ABB RobotStudio station: Box Sorting by Size v1.rspag

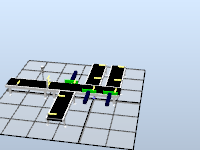
Station Box Sorting by Size v1 (saved by RobotStudio 21.4.9700.0)
Layout (positions relative to the parent item):
  - SUB010 [protected smart component, left out]
  - SUB020 [protected smart component, left out]
  - SUB050 [protected smart component, left out]
  - SUB040 [protected smart component, left out]
  - SUB030 [protected smart component, left out]
  - ProductInput [protected smart component, left out]
  - SUB600LightBeacon [protected smart component, left out]
  - OpcUaClient [smart component, from Components\OpcUaClient.rslib]
      properties: Status=Disconnected; ServerAddress=opc.tcp://localhost:4840; UseSecurity=false; AutoConnect=false; SignalConfiguration=NamespaceUri;IdentifierType;Identifier;ReadWrite;Signal;SignalType;Controller;Device
CODESYSSPV3/3S/IecVarAccess;String;|var|CODESYS Control Win V3 x64.Application.IOs.iSUB010_B1;Write;iSUB010_B1;Digital;;
CODESYSSPV3/3S/IecVarAccess;String;|var|CODESYS Control Win V3 x64.Application.IOs.iSUB010_B2;Write;iSUB010_B2;Digital;;
CODESYSSPV3/3S/IecVarAccess;String;|var|CODESYS Control Win V3 x64.Application.IOs.iSUB010_B3;Write;iSUB010_B3;Digital;;
CODESYSSPV3/3S/IecVarAccess;String;|var|CODESYS Control Win V3 x64.Application.IOs.iSUB010_B4;Write;iSUB010_B4;Digital;;
CODESYSSPV3/3S/IecVarAccess;String;|var|CODESYS Control Win V3 x64.Application.IOs.iSUB020_B1;Write;iSUB020_B1;Digital;;
CODESYSSPV3/3S/IecVarAccess;String;|var|CODESYS Control Win V3 x64.Application.IOs.iSUB020_B2;Write;iSUB020_B2;Digital;;
CODESYSSPV3/3S/IecVarAccess;String;|var|CODESYS Control Win V3 x64.Application.IOs.iSUB020_B3;Write;iSUB020_B3;Digital;;
CODESYSSPV3/3S/IecVarAccess;String;|var|CODESYS Control Win V3 x64.Application.IOs.iSUB030_B1;Write;iSUB030_B1;Digital;;
CODESYSSPV3/3S/IecVarAccess;String;|var|CODESYS Control Win V3 x64.Application.IOs.iSUB030_B2;Write;iSUB030_B2;Digital;;
CODESYSSPV3/3S/IecVarAccess;String;|var|CODESYS Control Win V3 x64.Application.IOs.iSUB030_C1_B1;Write;iSUB030_C1_B1;Digital;;
CODESYSSPV3/3S/IecVarAccess;String;|var|CODESYS Control Win V3 x64.Application.IOs.iSUB040_B1;Write;iSUB040_B1;Digital;;
CODESYSSPV3/3S/IecVarAccess;String;|var|CODESYS Control Win V3 x64.Application.IOs.iSUB040_B2;Write;iSUB040_B2;Digital;;
CODESYSSPV3/3S/IecVarAccess;String;|var|CODESYS Control Win V3 x64.Application.IOs.iSUB040_C1_B1;Write;iSUB040_C1_B1;Digital;;
CODESYSSPV3/3S/IecVarAccess;String;|var|CODESYS Control Win V3 x64.Application.IOs.iSUB050_B1;Write;iSUB050_B1;Digital;;
CODESYSSPV3/3S/IecVarAccess;String;|var|CODESYS Control Win V3 x64.Application.IOs.iSUB050_B2;Write;iSUB050_B2;Digital;;
CODESYSSPV3/3S/IecVarAccess;String;|var|CODESYS Control Win V3 x64.Application.IOs.iSUB050_C1_B1;Write;iSUB050_C1_B1;Digital;;
CODESYSSPV3/3S/IecVarAccess;String;|var|CODESYS Control Win V3 x64.Application.IOs.oSUB000_H4;Read;oSUB000_H4;Digital;;
CODESYSSPV3/3S/IecVarAccess;String;|var|CODESYS Control Win V3 x64.Application.IOs.oSUB000_H5;Read;oSUB000_H5;Digital;;
CODESYSSPV3/3S/IecVarAccess;String;|var|CODESYS Control Win V3 x64.Application.IOs.oSUB000_H6;Read;oSUB000_H6;Digital;;
CODESYSSPV3/3S/IecVarAccess;String;|var|CODESYS Control Win V3 x64.Application.IOs.oSUB010_K1;Read;oSUB010_K1;Digital;;
CODESYSSPV3/3S/IecVarAccess;String;|var|CODESYS Control Win V3 x64.Application.IOs.oSUB020_K1;Read;oSUB020_K1;Digital;;
CODESYSSPV3/3S/IecVarAccess;String;|var|CODESYS Control Win V3 x64.Application.IOs.oSUB030_K1;Read;oSUB030_K1;Digital;;
CODESYSSPV3/3S/IecVarAccess;String;|var|CODESYS Control Win V3 x64.Application.IOs.oSUB030_Y1;Read;oSUB030_Y1;Digital;;
CODESYSSPV3/3S/IecVarAccess;String;|var|CODESYS Control Win V3 x64.Application.IOs.oSUB040_K1;Read;oSUB040_K1;Digital;;
CODESYSSPV3/3S/IecVarAccess;String;|var|CODESYS Control Win V3 x64.Application.IOs.oSUB040_Y1;Read;oSUB040_Y1;Digital;;
CODESYSSPV3/3S/IecVarAccess;String;|var|CODESYS Control Win V3 x64.Application.IOs.oSUB050_K1;Read;oSUB050_K1;Digital;;
CODESYSSPV3/3S/IecVarAccess;String;|var|CODESYS Control Win V3 x64.Application.IOs.oSUB050_Y1;Read;oSUB050_Y1;Digital;;

  - SUB030Cylinder [protected smart component, left out]
  - SUB040Cylinder [protected smart component, left out]
  - SUB050Cylinder [protected smart component, left out]
  - Sensors [graphiccomponentgroup]
    - SUB010_B1 [protected smart component, left out]
    - SUB020_B1 [protected smart component, left out]
    - SUB020_B2 [protected smart component, left out]
    - SUB020_B3 [protected smart component, left out]
    - SUB030_B1 [protected smart component, left out]
    - SUB030_B2 [protected smart component, left out]
    - SUB040_B1 [protected smart component, left out]
    - SUB040_B2 [protected smart component, left out]
    - SUB050_B1 [protected smart component, left out]
    - SUB050_B2 [protected smart component, left out]
    - SUB010_B2 [protected smart component, left out]
    - SUB010_B3 [protected smart component, left out]
    - SUB010_B4 [protected smart component, left out]
  - Products [graphiccomponentgroup] at (-205.17, 3131.27, 530.83) mm
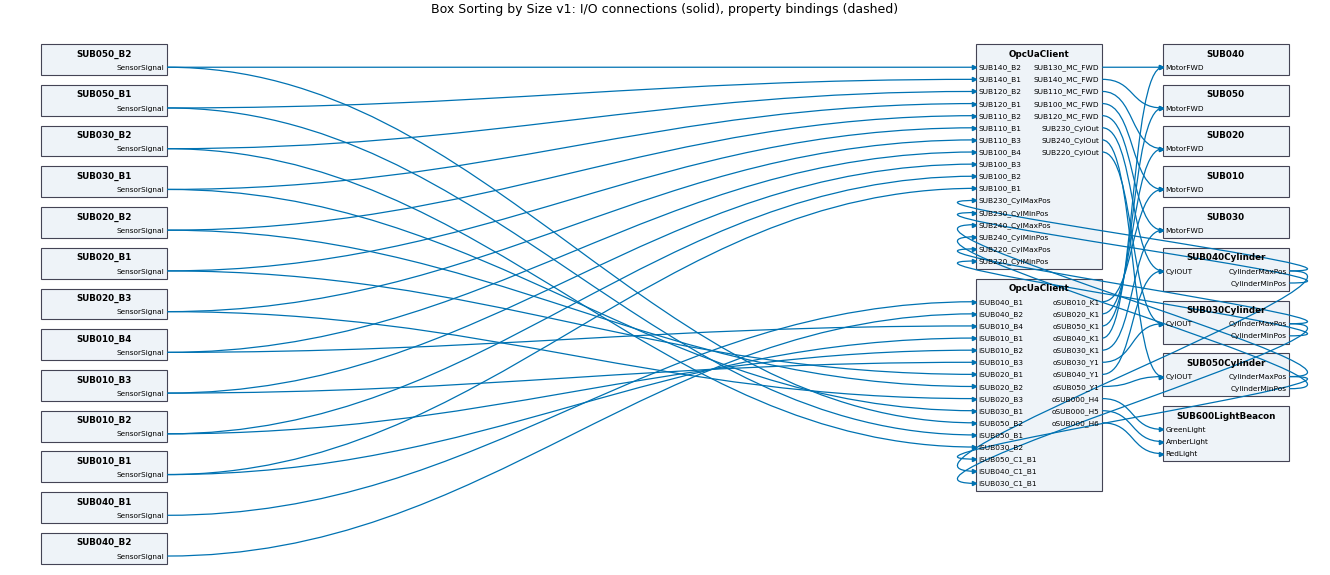
Station logic (signal -> signal, property => property):
  OpcUaClient.SUB130_MC_FWD -> SUB040.MotorFWD
  OpcUaClient.SUB140_MC_FWD -> SUB050.MotorFWD
  OpcUaClient.SUB110_MC_FWD -> SUB020.MotorFWD
  OpcUaClient.SUB100_MC_FWD -> SUB010.MotorFWD
  OpcUaClient.SUB120_MC_FWD -> SUB030.MotorFWD
  SUB050_B2.SensorSignal -> OpcUaClient.SUB140_B2
  SUB050_B1.SensorSignal -> OpcUaClient.SUB140_B1
  SUB030_B2.SensorSignal -> OpcUaClient.SUB120_B2
  SUB030_B1.SensorSignal -> OpcUaClient.SUB120_B1
  SUB020_B2.SensorSignal -> OpcUaClient.SUB110_B2
  SUB020_B1.SensorSignal -> OpcUaClient.SUB110_B1
  SUB020_B3.SensorSignal -> OpcUaClient.SUB110_B3
  SUB010_B4.SensorSignal -> OpcUaClient.SUB100_B4
  SUB010_B3.SensorSignal -> OpcUaClient.SUB100_B3
  SUB010_B2.SensorSignal -> OpcUaClient.SUB100_B2
  SUB010_B1.SensorSignal -> OpcUaClient.SUB100_B1
  OpcUaClient.SUB230_CylOut -> SUB040Cylinder.CylOUT
  SUB040Cylinder.CylinderMaxPos -> OpcUaClient.SUB230_CylMaxPos
  SUB040Cylinder.CylinderMinPos -> OpcUaClient.SUB230_CylMinPos
  OpcUaClient.SUB240_CylOut -> SUB050Cylinder.CylOUT
  SUB050Cylinder.CylinderMaxPos -> OpcUaClient.SUB240_CylMaxPos
  SUB050Cylinder.CylinderMinPos -> OpcUaClient.SUB240_CylMinPos
  SUB030Cylinder.CylinderMaxPos -> OpcUaClient.SUB220_CylMaxPos
  SUB030Cylinder.CylinderMinPos -> OpcUaClient.SUB220_CylMinPos
  OpcUaClient.SUB220_CylOut -> SUB030Cylinder.CylOUT
  SUB040_B1.SensorSignal -> OpcUaClient.iSUB040_B1
  SUB040_B2.SensorSignal -> OpcUaClient.iSUB040_B2
  OpcUaClient.oSUB010_K1 -> SUB010.MotorFWD
  OpcUaClient.oSUB020_K1 -> SUB020.MotorFWD
  OpcUaClient.oSUB050_K1 -> SUB050.MotorFWD
  OpcUaClient.oSUB040_K1 -> SUB040.MotorFWD
  OpcUaClient.oSUB030_K1 -> SUB030.MotorFWD
  SUB010_B4.SensorSignal -> OpcUaClient.iSUB010_B4
  SUB010_B1.SensorSignal -> OpcUaClient.iSUB010_B1
  SUB010_B2.SensorSignal -> OpcUaClient.iSUB010_B2
  SUB010_B3.SensorSignal -> OpcUaClient.iSUB010_B3
  SUB020_B1.SensorSignal -> OpcUaClient.iSUB020_B1
  SUB020_B2.SensorSignal -> OpcUaClient.iSUB020_B2
  SUB020_B3.SensorSignal -> OpcUaClient.iSUB020_B3
  SUB030_B1.SensorSignal -> OpcUaClient.iSUB030_B1
  SUB050_B2.SensorSignal -> OpcUaClient.iSUB050_B2
  SUB050_B1.SensorSignal -> OpcUaClient.iSUB050_B1
  SUB030_B2.SensorSignal -> OpcUaClient.iSUB030_B2
  SUB050Cylinder.CylinderMaxPos -> OpcUaClient.iSUB050_C1_B1
  SUB040Cylinder.CylinderMaxPos -> OpcUaClient.iSUB040_C1_B1
  SUB030Cylinder.CylinderMaxPos -> OpcUaClient.iSUB030_C1_B1
  OpcUaClient.oSUB030_Y1 -> SUB030Cylinder.CylOUT
  OpcUaClient.oSUB040_Y1 -> SUB040Cylinder.CylOUT
  OpcUaClient.oSUB050_Y1 -> SUB050Cylinder.CylOUT
  OpcUaClient.oSUB000_H4 -> SUB600LightBeacon.GreenLight
  OpcUaClient.oSUB000_H5 -> SUB600LightBeacon.AmberLight
  OpcUaClient.oSUB000_H6 -> SUB600LightBeacon.RedLight
